PROGRAM prgVarEffIO
VAR
	fbVar		: FB_VarInfo;
END_VAR

fbVar(
	bReadInfo:= , 
	eTMCFile:= eSelectTMCFile.eUseTMCFile, 
	eSavePositionTMCFile:= eSavePositionOnPLC.ePostionC, 
	udiCounterFoundVariables=> , 
	bError=> , 
	bBusy=> , 
	byProgress=> , 
	udiErrorCodeOut=> , 
	eErrorVarInfo_Out=> , 
	sVarWithError=> );
fbVar();
fbVar();

END_PROGRAM

(* stored: Version 1.1.0.1, ProductVersion 3.1.4024.12
   POU prgVarEffIO: Id {c92ea264-4e79-46c7-a0e1-0ebd92ac6f9d}, SpecialFunc None *)
